FUNCTION_BLOCK Safety1
VAR_INPUT
END_VAR
VAR_OUTPUT
END_VAR
VAR
	MaxRotationPosition: INT := 555;
	MaxLiftingPosition: INT := 270;
	MaxExtensionPosition: INT := 445;
	MaxGripPosition: INT := 170;
END_VAR

// Safety for Rotation:
IF Automatic.RotationPositionCurrent >= MaxRotationPosition AND NOT IO.ButtonLowerLeft AND NOT IO.MotorRotationDirection = 1 THEN
	Automatic.SafetyRON := TRUE;
	IO.MotorRotation := 0;
	IF Automatic.RotationPositionCurrent >= MaxRotationPosition THEN
		Automatic.RotationPositionCurrent := MaxRotationPosition;
	END_IF
	//Automatic.MotorR.CurrentlyMoving := FALSE;
	Automatic.RCurrentlyMoving := FALSE;
END_IF
IF IO.MotorRotationDirection = 0 THEN
	Automatic.SafetyRON := FALSE;
END_IF
IF IO.EndRotationSensor THEN
	IF IO.MotorRotationDirection = 0 THEN
		Automatic.SafetyRON := FALSE;
	ELSE
		Automatic.SafetyRON := TRUE;
		Automatic.RotationPositionCurrent := 0;
		Automatic.RotationPositionAuto := 0;
		//Automatic.MotorR.CurrentlyMoving := FALSE;
		Automatic.RCurrentlyMoving := FALSE;
	END_IF
END_IF

// Safety for Lifting:
IF Automatic.LiftingPositionCurrent >= MaxLiftingPosition AND NOT IO.ButtonLowerLeft AND NOT IO.MotorLiftingDirection = 1 THEN
	Automatic.SafetyLON := TRUE;
	IO.MotorLifting := 0;
	IF Automatic.LiftingPositionCurrent >= MaxLiftingPosition THEN
		Automatic.LiftingPositionCurrent := MaxLiftingPosition;
	END_IF
	//Automatic.MotorL.CurrentlyMoving := FALSE;
	Automatic.LCurrentlyMoving := FALSE;
END_IF
IF IO.MotorLiftingDirection = 0 THEN
	Automatic.SafetyLON := FALSE;
END_IF
IF IO.EndLiftingSensor THEN
	IF IO.MotorLiftingDirection = 0 THEN
		Automatic.SafetyLON := FALSE;
	ELSE
		Automatic.SafetyLON := TRUE;
		Automatic.LiftingPositionCurrent := 0;
		Automatic.LiftingPositionAuto := 0;
		//Automatic.MotorL.CurrentlyMoving := FALSE;
		Automatic.RCurrentlyMoving := FALSE;
	END_IF
END_IF

// Safety for Extension:
IF Automatic.ExtensionPositionCurrent >= MaxExtensionPosition AND NOT IO.ButtonLowerLeft AND NOT IO.MotorExtensionDirection = 1 THEN
	Automatic.SafetyEON := TRUE;
	IO.MotorExtension := 0;
	IF Automatic.ExtensionPositionCurrent >= MaxExtensionPosition THEN
		Automatic.ExtensionPositionCurrent := MaxExtensionPosition;
	END_IF
	//Automatic.MotorE.CurrentlyMoving := FALSE;
	Automatic.ECurrentlyMoving := FALSE;
END_IF
IF IO.MotorExtensionDirection = 0 THEN
	Automatic.SafetyEON := FALSE;
END_IF
IF IO.EndExtensionSensor THEN
	IF IO.MotorExtensionDirection = 0 THEN
		Automatic.SafetyEON := FALSE;
	ELSE
		Automatic.SafetyEON := TRUE;
		Automatic.ExtensionPositionCurrent := 0;
		Automatic.ExtensionPositionAuto := 0;
		//Automatic.MotorE.CurrentlyMoving := FALSE;
		Automatic.ECurrentlyMoving := FALSE;
	END_IF
END_IF

// Safety for Grip:
IF Automatic.GripPositionCurrent >= MaxGripPosition AND NOT IO.ButtonLowerLeft AND IO.MotorGripDirection = 0 THEN
	Automatic.SafetyGON := TRUE;
	IO.MotorGrip := 0;
	IF Automatic.GripPositionCurrent >= MaxGripPosition THEN
		Automatic.GripPositionCurrent := MaxGripPosition;
	END_IF
	//Automatic.GCurrentlyMoving := FALSE;
	Automatic.GCurrentlyMoving := FALSE;
END_IF
IF IO.MotorGripDirection = 1 THEN
	Automatic.SafetyGON := FALSE;
END_IF
IF IO.EndGripSensor THEN
	IF IO.MotorGripDirection = 0 THEN
		Automatic.SafetyGON := FALSE;
	ELSE
		Automatic.SafetyGON := TRUE;
		Automatic.GripPositionCurrent := 0;
		Automatic.GripPositionAuto := 0;
		//Automatic.GCurrentlyMoving := FALSE;
		Automatic.GCurrentlyMoving := FALSE;
	END_IF
END_IF

END_FUNCTION_BLOCK

(* stored: Version 1.1.0.1, ProductVersion 3.1.4024.13
   POU Safety1: Id {5dafd35d-1bf3-4cf6-972b-beee4c406310}, SpecialFunc None *)
